FUNCTION_BLOCK Eigenvalue2x2 (* Composite FB wrapping other FBs *)
  (* Standard: 61499-2; Description: Part of ellipse fitting method, to find eigenvalue. This block are specifically in use of ellipse fitting method, which doesn't generally exported. *)
  (* Version 1.0, 2020-08-19, Candra Wardaya, UGM *)
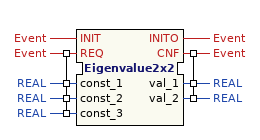
  EVENT_INPUT
    INIT; (* Initialization Request *)
    REQ WITH const_1, const_2, const_3; (* Normal Execution Request *)
  END_EVENT
  EVENT_OUTPUT
    INITO; (* Initialization Confirm *)
    CNF WITH val_1, val_2; (* Execution Confirmation *)
  END_EVENT
  VAR_INPUT
    const_1 : REAL; (* Single Real Input *)
    const_2 : REAL; (* Single Real Input *)
    const_3 : REAL; (* Single Real Input *)
  END_VAR
  VAR_OUTPUT
    val_1 : REAL; (* Single Real Output *)
    val_2 : REAL;
  END_VAR
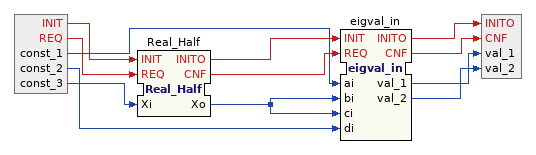
  FBS
    Real_Half : Real_Half;
    eigval_in : eigval_in;
  END_FBS
  EVENT_CONNECTIONS
    REQ TO Real_Half.REQ;
    INIT TO Real_Half.INIT;
    Real_Half.INITO TO eigval_in.INIT;
    Real_Half.CNF TO eigval_in.REQ;
    eigval_in.INITO TO INITO;
    eigval_in.CNF TO CNF;
  END_CONNECTIONS
  DATA_CONNECTIONS
    const_3 TO Real_Half.Xi;
    const_1 TO eigval_in.ai;
    Real_Half.Xo TO eigval_in.bi;
    Real_Half.Xo TO eigval_in.ci;
    const_2 TO eigval_in.di;
    eigval_in.val_1 TO val_1;
    eigval_in.val_2 TO val_2;
  END_CONNECTIONS
END_FUNCTION_BLOCK
